// TwinCAT 3 PLC project PLC1
// ProgramVersion: 3.1.4023.0
// libraries:
//   Tc2_Standard, * (Beckhoff Automation GmbH)
//   Tc2_System, * (Beckhoff Automation GmbH)
//   Tc2_Utilities, * (Beckhoff Automation GmbH)
//   Tc3_Module, * (Beckhoff Automation GmbH)
// project tree:
//   DUTs/ ChannelGuid.TcDUT, GuidCombo.TcDUT
//   GVLs/ GVL.TcGVL
//   / PlcTask.TcTTO
//   POUs/ Channel.TcPOU, Dictionary_I_Voltage.TcPOU, I_Voltage.TcIO, MAIN.TcPOU
// real-time tasks:
//   TASK PlcTask: cycle T#10ms, priority 20, ADS port 350

CONFIGURATION PLC1
    RESOURCE PLC ON TwinCAT3
        TASK PlcTask(INTERVAL := T#10ms, PRIORITY := 20);
        PROGRAM MAIN WITH PlcTask : MAIN;
    END_RESOURCE
END_CONFIGURATION

// ---- DUTs/ChannelGuid.TcDUT
TYPE ChannelGuid :
UNION
    GuidCombo : GuidCombo;
    GuidValue : DWORD;
END_UNION
END_TYPE

// ---- DUTs/GuidCombo.TcDUT
TYPE GuidCombo :
STRUCT
    TerminalAddress : WORD;
    ChannelNumber : WORD;
END_STRUCT
END_TYPE

// ---- GVLs/GVL.TcGVL
{attribute 'qualified_only'}
VAR_GLOBAL CONSTANT
    DICTIONARY_UPPER_BOUND : INT := 4;
END_VAR

// ---- POUs/I_Voltage.TcIO
INTERFACE I_Voltage

PROPERTY GUID : DWORD
GET
END_GET
END_PROPERTY

PROPERTY Name : STRING
GET
END_GET
SET
END_SET
END_PROPERTY

END_INTERFACE

// ---- POUs/MAIN.TcPOU
PROGRAM MAIN
VAR
    ch1 : Channel(10,1);
    ch2 : Channel(10,2);
    ch3 : Channel(10,4);
    ch4 : Channel(11,1);
    ch5 : Channel(11,2);
    ch6 : Channel(11,3);
    ch7 : I_Voltage;
    chKey : DWORD;
    channels : Dictionary_I_Voltage;
    addCh : BOOL;
    getCh : BOOL;
    getChAt : BOOL;
    removeCh : BOOL;
    clear : BOOL;
    result : BOOL;
    index : INT;
END_VAR

IF addCh THEN
    addCh := FALSE;
    result := channels.TryAdd(ch1);
    result := channels.TryAdd(ch2);
    result := channels.TryAdd(ch3);
    result := channels.TryAdd(ch4);
    result := channels.TryAdd(ch5);
END_IF

IF getCh THEN
    getCh := FALSE;
    result := channels.TryGet(10,4,item=>ch7);
END_IF

IF getChAt THEN
    getChAt := FALSE;
    result := channels.TryGetAt(index,key=>chKey,item=>ch7);
END_IF

IF removeCh THEN
    removeCh := FALSE;
    channels.Remove(10,4);
END_IF

IF clear THEN
    clear := FALSE;
    channels.Clear();
END_IF

END_PROGRAM

// ---- POUs/Channel.TcPOU
FUNCTION_BLOCK Channel IMPLEMENTS I_Voltage
VAR_INPUT
END_VAR
VAR_OUTPUT
END_VAR
VAR
    _terminalAddress : WORD;
    _channelNumber : WORD;
    _guid : ChannelGuid;
    _name : STRING;
END_VAR

METHOD FB_init : BOOL
VAR_INPUT
	bInitRetains : BOOL; // if TRUE, the retain variables are initialized (warm start / cold start)
	bInCopyCode : BOOL;  // if TRUE, the instance afterwards gets moved into the copy code (online change)
    termianlAddress : WORD;
    channelNumber : WORD;
END_VAR
_terminalAddress := termianlAddress;
_channelNumber := channelNumber;
_guid.GuidCombo.ChannelNumber := _channelNumber;
_guid.GuidCombo.TerminalAddress := _terminalAddress;
END_METHOD

PROPERTY GUID : DWORD
GET
GUID := _guid.GuidValue;
END_GET
END_PROPERTY

PROPERTY Name : STRING
GET
Name := _name;
END_GET
SET
_name := Name;
END_SET
END_PROPERTY

END_FUNCTION_BLOCK

// ---- POUs/Dictionary_I_Voltage.TcPOU
FUNCTION_BLOCK Dictionary_I_Voltage
VAR_INPUT
END_VAR
VAR_OUTPUT
END_VAR
VAR
    _dataPool : ARRAY[0..GVL.DICTIONARY_UPPER_BOUND] OF I_Voltage;
    _hashTableEntries : ARRAY[0..GVL.DICTIONARY_UPPER_BOUND] OF Tc2_Utilities.T_HashTableEntry;
    _hashTable : Tc2_Utilities.FB_HashTableCtrl;
    _hashTableHandler : Tc2_Utilities.T_HHASHTABLE;
END_VAR

METHOD Clear
VAR
    i : INT;
END_VAR
F_CreateHashTableHnd(ADR(_hashTableEntries), SIZEOF(_hashTableEntries), _hashTableHandler ); //Intialize table handle
_hashTable.A_Reset(hTable:=_hashTableHandler);
FOR i:=0 TO GVL.DICTIONARY_UPPER_BOUND DO
    _dataPool[i] := 0;
END_FOR
END_METHOD

METHOD FB_init : BOOL
VAR_INPUT
	bInitRetains : BOOL; // if TRUE, the retain variables are initialized (warm start / cold start)
	bInCopyCode : BOOL;  // if TRUE, the instance afterwards gets moved into the copy code (online change)
END_VAR
F_CreateHashTableHnd(ADR(_hashTableEntries), SIZEOF(_hashTableEntries), _hashTableHandler ); //Intialize table handle
END_METHOD

METHOD GetCount : INT
GetCount := UDINT_TO_INT(_hashTableHandler.nCount);
END_METHOD

METHOD Remove
VAR_INPUT
    terminalAddress : WORD;
    channelNumber : WORD;
END_VAR
VAR
    itemGuid : ChannelGuid;
    entryValuePtr : POINTER TO I_Voltage;
END_VAR
itemGuid.GuidCombo.TerminalAddress := terminalAddress;
itemGuid.GuidCombo.ChannelNumber := channelNumber;
_hashTable.A_Remove(key:=itemGuid.GuidValue, hTable:=_hashTableHandler, getValue=>entryValuePtr);
IF _hashTable.bOk THEN
	entryValuePtr^ := 0;
END_IF
END_METHOD

METHOD TryAdd : BOOL
VAR_INPUT
    item : I_Voltage;
END_VAR
VAR
    newEntryPtr	: POINTER TO T_HashTableEntry;
	indexOfnewEntry	: ULINT;
END_VAR
_hashTable.A_Add(hTable:=_hashTableHandler, key:=item.GUID, putValue:=16#FFFFFFFF, getPosPtr=>newEntryPtr); //Just to get a proper Index, later we assign the real value
IF _hashTable.bOk THEN
	_hashTable.A_GetIndexAtPosPtr(hTable:=_hashTableHandler, putPosPtr:=newEntryPtr, getValue=>indexOfnewEntry);
	IF _hashTable.bOk THEN
		_dataPool[indexOfnewEntry] := item;
		_hashTable.A_Add(hTable:=_hashTableHandler, key:=item.GUID,putValue:=ADR(_dataPool[indexOfnewEntry]));
		IF _hashTable.bOk THEN
			TryAdd := TRUE;
		END_IF
	END_IF
END_IF
END_METHOD

METHOD TryGet : BOOL
VAR_INPUT
    terminalAddress : WORD;
    channelNumber : WORD;
END_VAR
VAR_OUTPUT
    item : I_Voltage;
END_VAR
VAR
    itemGuid : ChannelGuid;
    entryValuePtr : POINTER TO I_Voltage;
END_VAR
itemGuid.GuidCombo.TerminalAddress := terminalAddress;
itemGuid.GuidCombo.ChannelNumber := channelNumber;
_hashTable.A_Lookup(key:=itemGuid.GuidValue, hTable:=_hashTableHandler, getValue=>entryValuePtr);
IF _hashTable.bOk THEN
	item := entryValuePtr^;
    IF item<>0 THEN
        TryGet := TRUE;
	END_IF
END_IF
END_METHOD

METHOD TryGetAt : BOOL
VAR_INPUT
    index : INT;
END_VAR
VAR_OUTPUT
    key : DWORD;
    item : I_Voltage;
END_VAR
VAR
    entryPtr : POINTER TO T_HashTableEntry;
    entryValuePtr : POINTER TO I_Voltage;
    i : INT;
END_VAR
IF index<0 OR index>=GetCount() THEN
    TryGetAt := FALSE;
    RETURN;
END_IF
index := GetCount()-(index+1);

_hashTable.A_GetFirst(hTable:=_hashTableHandler, putPosPtr:=0, getValue=>entryValuePtr, getPosPtr=>entryPtr);
IF _hashTable.bOk THEN
    FOR i:=1 TO index DO
        _hashTable.A_GetNext(hTable:=_hashTableHandler, putPosPtr:=entryPtr, getValue=>entryValuePtr, getPosPtr=>entryPtr);
	END_FOR
    IF _hashTable.bOk THEN
        item := entryValuePtr^;
        key := entryPtr^.key;
        IF item<>0 THEN
            TryGetAt := TRUE;
        END_IF
	END_IF
END_IF
END_METHOD

END_FUNCTION_BLOCK
